{attribute 'GeneratedUsingTerminal: EK1122-0000-0018'}
{attribute addProperty BoxType "EK1122-0000-0018"}
{attribute addProperty Id "Beckhoff_EKxxxx_0080sub_EK1100EK1100_AB5A94672"}
{attribute addProperty CRC "1921036100"}
{attribute addProperty Size "2"}
TYPE Beckhoff_EKxxxx_0080EK1122_7280AF44 EXTENDS EK1122_AB5A9467 :
STRUCT
	{attribute addProperty Name "Beckhoff_EKxxxx_0080sub_EK1100"}
	Beckhoff_EKxxxx_0080sub_EK1100 : EK1100_AB5A9467;
END_STRUCT
END_TYPE

(* stored: Version 1.2.0.0, ProductVersion 3.1.4024.9
   DUT Beckhoff_EKxxxx_0080EK1122_7280AF44: Id {3dc9e995-ab2e-4e64-9c6e-c35ad2416e8f} *)
